// TIA Portal V19 export
FUNCTION_BLOCK "Coilcar_FB"   // FB96, LAD
TITLE = COIL CAR
// stored: MemoryReserve 100, SetENOAutomatically false
   VAR_INPUT
      AreaInterface : "AreaInterface";
      ZSI : "udt_ZoneSafetyInterface";
      DSI : Struct
         Move : "udt_DeviceSafetyInterface";
         LIft : "udt_DeviceSafetyInterface";
      END_STRUCT;
      Drive : "TAx_DriveInterface";
      HW_ID_TEL1 : HW_SUBMODULE;
      DataIn : Struct
         Supports_Ls_FixPoleLeft_Plugged : Bool;
         Supports_Ls_FixPoleRight_Plugged : Bool;
         Supports_Ls_MobilePoleLeft_Plugged : Bool;
         Supports_Ls_MobilePoleRight_Plugged : Bool;
         Move_Ls_Outline : Bool;
         Move_Ls_Inline : Bool;
         Move_Ls_LowSpeedOutline : Bool;
         Move_Ls_LowSpeedInline : Bool;
         Move_Ls_CoilInserted : Bool;   // TRUE = Movable supprts must be closed
         Move : "SpeedMachine_DataIn";
         Lift1 : "ValveMachine_DataIn";
         Lift2 : "ValveMachine_DataIn";
      END_STRUCT;
      CIn : Struct
         PressureRunning : Bool;
      END_STRUCT;
      Config : Struct
         LsStopDelayON { ExternalAccessible := 'False'; ExternalVisible := 'False'; ExternalWritable := 'False'} : Time := T#100ms;
         LsStopDelayOFF { ExternalAccessible := 'False'; ExternalVisible := 'False'; ExternalWritable := 'False'} : Time := T#200ms;
         Move : "SpeedMachine_Config";
         Lift1 : "ValveMachine_Config";
         Lift2 : "ValveMachine_Config";
      END_STRUCT;
   END_VAR
   VAR_OUTPUT
      MachineInterface : "MachineInterface";
      DataOut : Struct
         Move : "SpeedMachine_DataOut";
         Lift1 : "ValveMachine_DataOut";
         Lift2 : "ValveMachine_DataOut";
      END_STRUCT;
      COut : Struct
         IsInline : Bool;
         IsOutline : Bool;
         Move : "SpeedMachine_COut";
         Lift1 : "ValveMachine_COut";
         Lift2 : "ValveMachine_COut";
      END_STRUCT;
   END_VAR
   VAR_IN_OUT
      PersistentValues : Struct
         Move : "SpeedMachine_Par";
      END_STRUCT;
   END_VAR
   VAR
      Sts : Struct
         Move : Struct
            LowSpeedInline : Bool;
            LowSpeedOutline : Bool;
            IsInline : Bool;
            IsOutline : Bool;
            Inline_Cnd : Bool;
            Outline_Cnd : Bool;
            ReductionRatio : LReal;
         END_STRUCT;
         Free : Bool;
      END_STRUCT;
      Alarm : Struct
         Move_UnvalidStateLsInOut : Bool;
         Move_UnvalidStateLsLow : Bool;
         Move : "SpeedMachine_Alr";
         Lift1 : "ValveAlr";
         Lift2 : "ValveAlr";
      END_STRUCT;
      Warning : Struct
         Move : "SpeedMachine_Wng";
         Lift1 { ExternalAccessible := 'False'; ExternalVisible := 'False'; ExternalWritable := 'False'} : "ValveMachine_Wng";
         Lift2 { ExternalAccessible := 'False'; ExternalVisible := 'False'; ExternalWritable := 'False'} : "ValveMachine_Wng";
         NotOutline : Bool;
         Supports_FixPolesNotPlugged : Bool;
         Supports_MobilePolesNotPlugged : Bool;
      END_STRUCT;
      Move : "SpeedMachine_FB";
      Lift1 : "ValveMachine_FB";
      Lift2 : "ValveMachine_FB";
      TON_OutlinePos_DelayON : IEC_TIMER;
      TON_OutlinePos_DelayOFF : IEC_TIMER;
      TON_InlinePos_DelayON : IEC_TIMER;
      TON_InlinePos_DelayOFF : IEC_TIMER;
      pippo { S7_SetPoint := 'True'} : IEC_TIMER;
   END_VAR
   VAR_TEMP   // added for the SCL form of the ladder/FBD networks
      _w1 : Bool;
   END_VAR
BEGIN

REGION Network 1 (SCL): Reset alarms command

   IF  #AreaInterface.RstAlarms THEN
       // Alarms
       #Alarm.Move_UnvalidStateLsInOut := FALSE;
       #Alarm.Move_UnvalidStateLsLow := FALSE;



   END_IF;
END_REGION

REGION Network 2: >
END_REGION

REGION Network 3: <<< MOVE >>>
END_REGION

REGION Network 4: Alarm: Invalid state of inline/outline limit switches
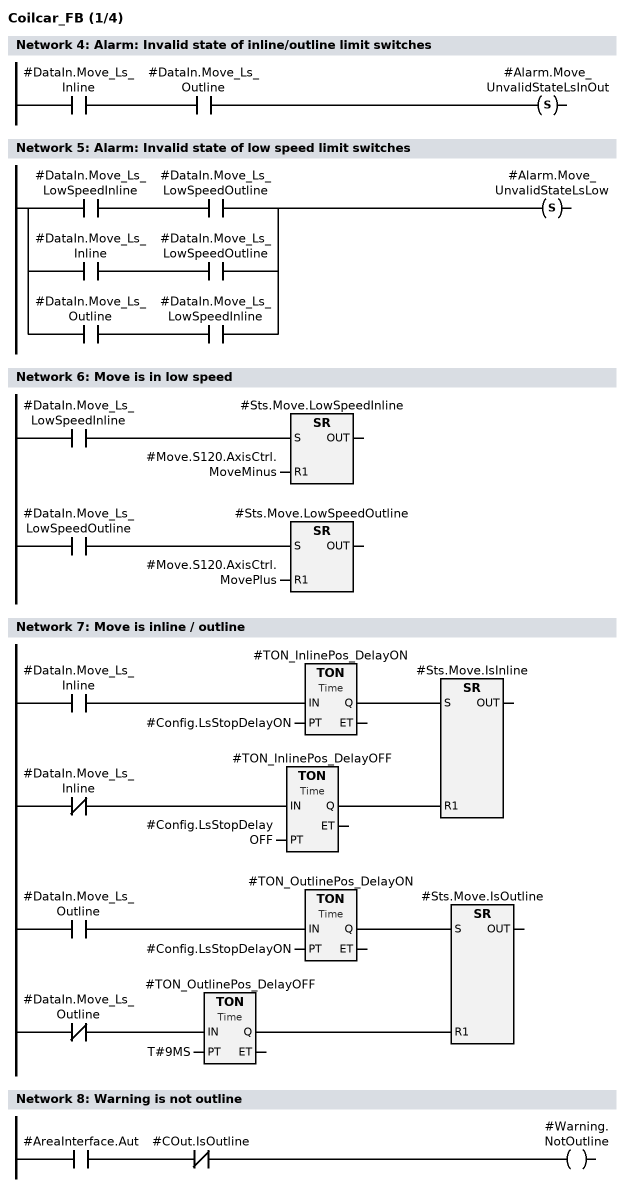
   RUNG wire#powerrail
      Contact( #DataIn.Move_Ls_Inline )
      Contact( #DataIn.Move_Ls_Outline )
      S_Coil( #Alarm.Move_UnvalidStateLsInOut )
   END_RUNG
   // the same network as SCL:
   IF #DataIn.Move_Ls_Inline AND #DataIn.Move_Ls_Outline THEN
       #Alarm.Move_UnvalidStateLsInOut := TRUE;
   END_IF;
END_REGION

REGION Network 5: Alarm: Invalid state of low speed limit switches
   RUNG wire#powerrail
      Contact( #DataIn.Move_Ls_LowSpeedInline )
      Contact( #DataIn.Move_Ls_LowSpeedOutline )
      wire#w1
      S_Coil( #Alarm.Move_UnvalidStateLsLow )
   END_RUNG
   RUNG wire#powerrail
      Contact( #DataIn.Move_Ls_Inline )
      Contact( #DataIn.Move_Ls_LowSpeedOutline )
   END_RUNG wire#w1
   RUNG wire#powerrail
      Contact( #DataIn.Move_Ls_Outline )
      Contact( #DataIn.Move_Ls_LowSpeedInline )
   END_RUNG wire#w1
   // the same network as SCL:
   IF (#DataIn.Move_Ls_LowSpeedInline AND #DataIn.Move_Ls_LowSpeedOutline) OR (#DataIn.Move_Ls_Inline AND #DataIn.Move_Ls_LowSpeedOutline) OR (#DataIn.Move_Ls_Outline AND #DataIn.Move_Ls_LowSpeedInline) THEN
       #Alarm.Move_UnvalidStateLsLow := TRUE;
   END_IF;
END_REGION

REGION Network 6: Move is in low speed
   RUNG wire#powerrail
      Contact( #DataIn.Move_Ls_LowSpeedInline )
      S_SR(operand := #Sts.Move.LowSpeedInline, r1 := #Move.S120.AxisCtrl.MoveMinus)
   END_RUNG
   RUNG wire#powerrail
      Contact( #DataIn.Move_Ls_LowSpeedOutline )
      S_SR(operand := #Sts.Move.LowSpeedOutline, r1 := #Move.S120.AxisCtrl.MovePlus)
   END_RUNG
   // the same network as SCL:
   IF #DataIn.Move_Ls_LowSpeedInline THEN
       #Sts.Move.LowSpeedInline := TRUE;   // SR flip-flop
   END_IF;
   IF #Move.S120.AxisCtrl.MoveMinus THEN #Sts.Move.LowSpeedInline := FALSE; END_IF;
   IF #DataIn.Move_Ls_LowSpeedOutline THEN
       #Sts.Move.LowSpeedOutline := TRUE;   // SR flip-flop
   END_IF;
   IF #Move.S120.AxisCtrl.MovePlus THEN #Sts.Move.LowSpeedOutline := FALSE; END_IF;
END_REGION

REGION Network 7: Move is inline / outline
   RUNG wire#powerrail
      Contact( #DataIn.Move_Ls_Inline )
      { S7_Templates := "time_type := Time" } #TON_InlinePos_DelayON.TON(pt := #Config.LsStopDelayON, et =>)
      S_SR(operand := #Sts.Move.IsInline, r1 := wire#w1)
   END_RUNG
   RUNG wire#powerrail
      I_Contact( #DataIn.Move_Ls_Inline )
      { S7_Templates := "time_type := Time" } #TON_InlinePos_DelayOFF.TON(pt := #Config.LsStopDelayOFF, et =>)
   END_RUNG wire#w1
   RUNG wire#powerrail
      Contact( #DataIn.Move_Ls_Outline )
      { S7_Templates := "time_type := Time" } #TON_OutlinePos_DelayON.TON(pt := #Config.LsStopDelayON, et =>)
      S_SR(operand := #Sts.Move.IsOutline, r1 := wire#w2)
   END_RUNG
   RUNG wire#powerrail
      I_Contact( #DataIn.Move_Ls_Outline )
      { S7_Templates := "time_type := Time" } #TON_OutlinePos_DelayOFF.TON(pt := T#9MS, et =>)
   END_RUNG wire#w2
   // the same network as SCL:
   #TON_InlinePos_DelayON.TON(IN := #DataIn.Move_Ls_Inline, PT := #Config.LsStopDelayON);
   #TON_InlinePos_DelayOFF.TON(IN := NOT #DataIn.Move_Ls_Inline, PT := #Config.LsStopDelayOFF);
   IF #TON_InlinePos_DelayON.Q THEN
       #Sts.Move.IsInline := TRUE;   // SR flip-flop
   END_IF;
   IF #TON_InlinePos_DelayOFF.Q THEN #Sts.Move.IsInline := FALSE; END_IF;
   #TON_OutlinePos_DelayON.TON(IN := #DataIn.Move_Ls_Outline, PT := #Config.LsStopDelayON);
   #TON_OutlinePos_DelayOFF.TON(IN := NOT #DataIn.Move_Ls_Outline, PT := T#9MS);
   IF #TON_OutlinePos_DelayON.Q THEN
       #Sts.Move.IsOutline := TRUE;   // SR flip-flop
   END_IF;
   IF #TON_OutlinePos_DelayOFF.Q THEN #Sts.Move.IsOutline := FALSE; END_IF;
END_REGION

REGION Network 8: Warning is not outline
   RUNG wire#powerrail
      Contact( #AreaInterface.Aut )
      I_Contact( #COut.IsOutline )
      Coil( #Warning.NotOutline )
   END_RUNG
   // the same network as SCL:
   #Warning.NotOutline := #AreaInterface.Aut AND NOT #COut.IsOutline;
END_REGION

REGION Network 9: Warnings for missing rotation conditions
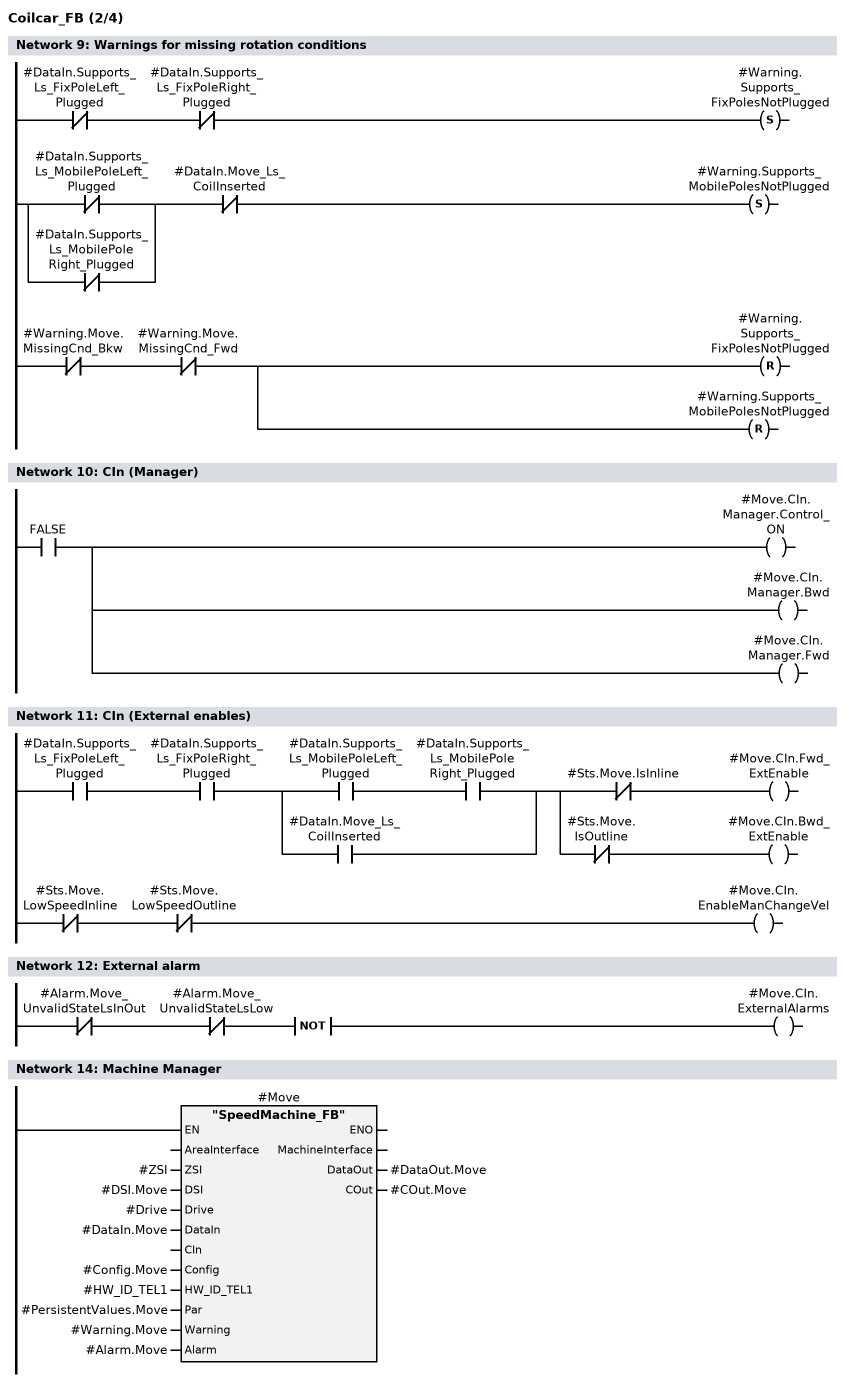
   RUNG wire#powerrail
      I_Contact( #DataIn.Supports_Ls_FixPoleLeft_Plugged )
      I_Contact( #DataIn.Supports_Ls_FixPoleRight_Plugged )
      S_Coil( #Warning.Supports_FixPolesNotPlugged )
   END_RUNG
   RUNG wire#powerrail
      I_Contact( #DataIn.Supports_Ls_MobilePoleLeft_Plugged )
      wire#w1
      I_Contact( #DataIn.Move_Ls_CoilInserted )
      S_Coil( #Warning.Supports_MobilePolesNotPlugged )
   END_RUNG
   RUNG wire#powerrail
      I_Contact( #DataIn.Supports_Ls_MobilePoleRight_Plugged )
   END_RUNG wire#w1
   RUNG wire#powerrail
      I_Contact( #Warning.Move.MissingCnd_Bkw )
      I_Contact( #Warning.Move.MissingCnd_Fwd )
      wire#w2
      R_Coil( #Warning.Supports_FixPolesNotPlugged )
   END_RUNG
   RUNG wire#w2
      R_Coil( #Warning.Supports_MobilePolesNotPlugged )
   END_RUNG
   // the same network as SCL:
   IF NOT #DataIn.Supports_Ls_FixPoleLeft_Plugged AND NOT #DataIn.Supports_Ls_FixPoleRight_Plugged THEN
       #Warning.Supports_FixPolesNotPlugged := TRUE;
   END_IF;
   IF (NOT #DataIn.Supports_Ls_MobilePoleLeft_Plugged OR NOT #DataIn.Supports_Ls_MobilePoleRight_Plugged) AND NOT #DataIn.Move_Ls_CoilInserted THEN
       #Warning.Supports_MobilePolesNotPlugged := TRUE;
   END_IF;
   IF NOT #Warning.Move.MissingCnd_Bkw AND NOT #Warning.Move.MissingCnd_Fwd THEN
       #Warning.Supports_FixPolesNotPlugged := FALSE;
       #Warning.Supports_MobilePolesNotPlugged := FALSE;
   END_IF;
END_REGION

REGION Network 10: CIn (Manager)
   RUNG wire#powerrail
      Contact( FALSE )
      wire#w1
      Coil( #Move.CIn.Manager.Control_ON )
   END_RUNG
   RUNG wire#w1
      Coil( #Move.CIn.Manager.Bwd )
   END_RUNG
   RUNG wire#w1
      Coil( #Move.CIn.Manager.Fwd )
   END_RUNG
   // the same network as SCL:
   #Move.CIn.Manager.Control_ON := FALSE;
   #Move.CIn.Manager.Bwd := FALSE;
   #Move.CIn.Manager.Fwd := FALSE;
END_REGION

REGION Network 11: CIn (External enables)
   RUNG wire#powerrail
      Contact( #DataIn.Supports_Ls_FixPoleLeft_Plugged )
      Contact( #DataIn.Supports_Ls_FixPoleRight_Plugged )
      wire#w1
      Contact( #DataIn.Supports_Ls_MobilePoleLeft_Plugged )
      Contact( #DataIn.Supports_Ls_MobilePoleRight_Plugged )
      wire#w2
      I_Contact( #Sts.Move.IsInline )
      Coil( #Move.CIn.Fwd_ExtEnable )
   END_RUNG
   RUNG wire#w1
      Contact( #DataIn.Move_Ls_CoilInserted )
   END_RUNG wire#w2
   RUNG wire#w2
      I_Contact( #Sts.Move.IsOutline )
      Coil( #Move.CIn.Bwd_ExtEnable )
   END_RUNG
   RUNG wire#powerrail
      I_Contact( #Sts.Move.LowSpeedInline )
      I_Contact( #Sts.Move.LowSpeedOutline )
      Coil( #Move.CIn.EnableManChangeVel )
   END_RUNG
   // the same network as SCL:
   #_w1 := #DataIn.Supports_Ls_FixPoleLeft_Plugged AND #DataIn.Supports_Ls_FixPoleRight_Plugged AND ((#DataIn.Supports_Ls_MobilePoleLeft_Plugged AND #DataIn.Supports_Ls_MobilePoleRight_Plugged) OR #DataIn.Move_Ls_CoilInserted);
   #Move.CIn.Fwd_ExtEnable := #_w1 AND NOT #Sts.Move.IsInline;
   #Move.CIn.Bwd_ExtEnable := #_w1 AND NOT #Sts.Move.IsOutline;
   #Move.CIn.EnableManChangeVel := NOT #Sts.Move.LowSpeedInline AND NOT #Sts.Move.LowSpeedOutline;
END_REGION

REGION Network 12: External alarm
   RUNG wire#powerrail
      I_Contact( #Alarm.Move_UnvalidStateLsInOut )
      I_Contact( #Alarm.Move_UnvalidStateLsLow )
      Not()
      Coil( #Move.CIn.ExternalAlarms )
   END_RUNG
   // the same network as SCL:
   #Move.CIn.ExternalAlarms := NOT (NOT #Alarm.Move_UnvalidStateLsInOut AND NOT #Alarm.Move_UnvalidStateLsLow);
END_REGION

REGION Network 13 (SCL): AreaInterface
   #Move.AreaInterface := #AreaInterface;

   #Move.AreaInterface.Man := #AreaInterface.Aut OR #AreaInterface.Man;
   #Move.AreaInterface.Aut := FALSE;
   #Move.AreaInterface.Cycle := FALSE;
END_REGION

REGION Network 14: Machine Manager
   RUNG wire#powerrail
      #Move(AreaInterface :=, ZSI := #ZSI, DSI := #DSI.Move, Drive := #Drive, DataIn := #DataIn.Move, CIn :=, Config := #Config.Move, HW_ID_TEL1 := #HW_ID_TEL1, Par := #PersistentValues.Move, Warning := #Warning.Move, Alarm := #Alarm.Move, MachineInterface =>, DataOut => #DataOut.Move, COut => #COut.Move)
   END_RUNG
   // the same network as SCL:
   #Move(ZSI := #ZSI,   // "SpeedMachine_FB"
         DSI := #DSI.Move,
         Drive := #Drive,
         DataIn := #DataIn.Move,
         Config := #Config.Move,
         HW_ID_TEL1 := #HW_ID_TEL1,
         Par := #PersistentValues.Move,
         Warning := #Warning.Move,
         Alarm := #Alarm.Move,
         DataOut => #DataOut.Move,
         COut => #COut.Move);
END_REGION

REGION Network 15: >
END_REGION

REGION Network 16: >
END_REGION

REGION Network 17: <<< LIFT 1 (REST = DOWN / WORK = UP)>>>
END_REGION

REGION Network 18: CIn (external enables)
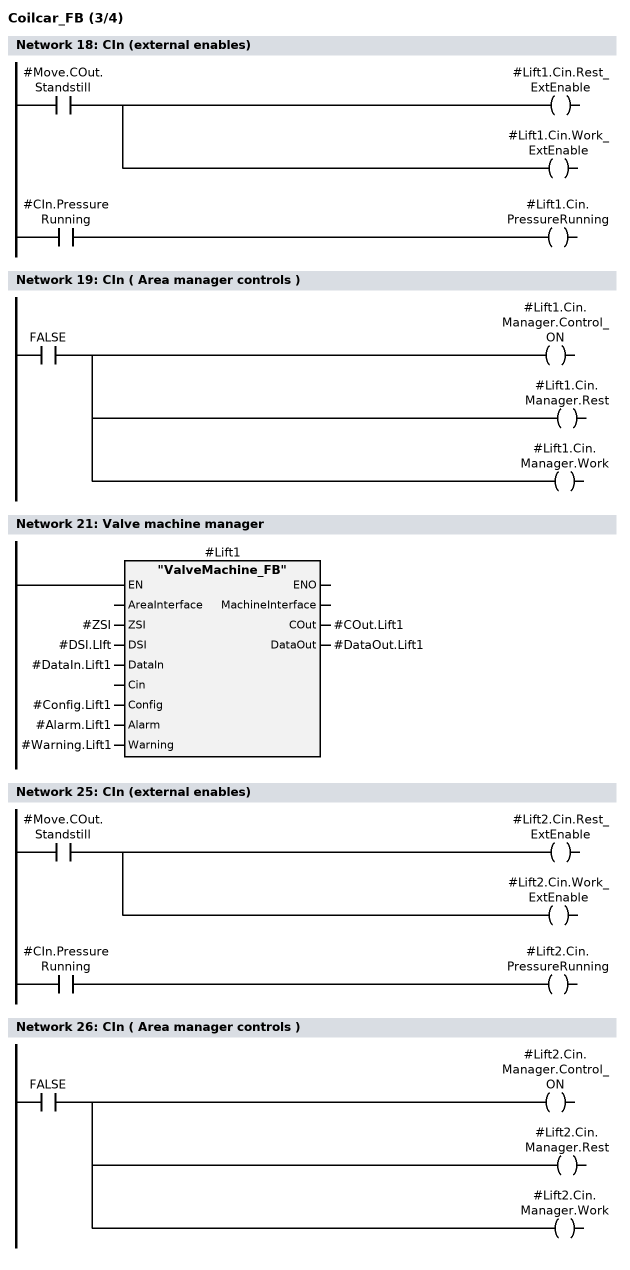
   RUNG wire#powerrail
      Contact( #Move.COut.Standstill )
      wire#w1
      Coil( #Lift1.Cin.Rest_ExtEnable )
   END_RUNG
   RUNG wire#w1
      Coil( #Lift1.Cin.Work_ExtEnable )
   END_RUNG
   RUNG wire#powerrail
      Contact( #CIn.PressureRunning )
      Coil( #Lift1.Cin.PressureRunning )
   END_RUNG
   // the same network as SCL:
   #Lift1.Cin.Rest_ExtEnable := #Move.COut.Standstill;
   #Lift1.Cin.Work_ExtEnable := #Move.COut.Standstill;
   #Lift1.Cin.PressureRunning := #CIn.PressureRunning;
END_REGION

REGION Network 19: CIn ( Area manager controls )
   RUNG wire#powerrail
      Contact( FALSE )
      wire#w1
      Coil( #Lift1.Cin.Manager.Control_ON )
   END_RUNG
   RUNG wire#w1
      Coil( #Lift1.Cin.Manager.Rest )
   END_RUNG
   RUNG wire#w1
      Coil( #Lift1.Cin.Manager.Work )
   END_RUNG
   // the same network as SCL:
   #Lift1.Cin.Manager.Control_ON := FALSE;
   #Lift1.Cin.Manager.Rest := FALSE;
   #Lift1.Cin.Manager.Work := FALSE;
END_REGION

REGION Network 20 (SCL): AreaInterface
   #Lift1.AreaInterface := #AreaInterface;

   #Lift1.AreaInterface.Man := #AreaInterface.Aut OR #AreaInterface.Man;
   #Lift1.AreaInterface.Aut := FALSE;
   #Lift1.AreaInterface.Cycle := FALSE;
END_REGION

REGION Network 21: Valve machine manager
   RUNG wire#powerrail
      #Lift1(AreaInterface :=, ZSI := #ZSI, DSI := #DSI.LIft, DataIn := #DataIn.Lift1, Cin :=, Config := #Config.Lift1, Alarm := #Alarm.Lift1, Warning := #Warning.Lift1, MachineInterface =>, COut => #COut.Lift1, DataOut => #DataOut.Lift1)
   END_RUNG
   // the same network as SCL:
   #Lift1(ZSI := #ZSI,   // "ValveMachine_FB"
          DSI := #DSI.LIft,
          DataIn := #DataIn.Lift1,
          Config := #Config.Lift1,
          Alarm := #Alarm.Lift1,
          Warning := #Warning.Lift1,
          COut => #COut.Lift1,
          DataOut => #DataOut.Lift1);
END_REGION

REGION Network 22: >
END_REGION

REGION Network 23: >
END_REGION

REGION Network 24: <<< LIFT 1 (REST = DOWN / WORK = UP)>>>
END_REGION

REGION Network 25: CIn (external enables)
   RUNG wire#powerrail
      Contact( #Move.COut.Standstill )
      wire#w1
      Coil( #Lift2.Cin.Rest_ExtEnable )
   END_RUNG
   RUNG wire#w1
      Coil( #Lift2.Cin.Work_ExtEnable )
   END_RUNG
   RUNG wire#powerrail
      Contact( #CIn.PressureRunning )
      Coil( #Lift2.Cin.PressureRunning )
   END_RUNG
   // the same network as SCL:
   #Lift2.Cin.Rest_ExtEnable := #Move.COut.Standstill;
   #Lift2.Cin.Work_ExtEnable := #Move.COut.Standstill;
   #Lift2.Cin.PressureRunning := #CIn.PressureRunning;
END_REGION

REGION Network 26: CIn ( Area manager controls )
   RUNG wire#powerrail
      Contact( FALSE )
      wire#w1
      Coil( #Lift2.Cin.Manager.Control_ON )
   END_RUNG
   RUNG wire#w1
      Coil( #Lift2.Cin.Manager.Rest )
   END_RUNG
   RUNG wire#w1
      Coil( #Lift2.Cin.Manager.Work )
   END_RUNG
   // the same network as SCL:
   #Lift2.Cin.Manager.Control_ON := FALSE;
   #Lift2.Cin.Manager.Rest := FALSE;
   #Lift2.Cin.Manager.Work := FALSE;
END_REGION

REGION Network 27 (SCL): AreaInterface
   #Lift2.AreaInterface := #AreaInterface;

   #Lift2.AreaInterface.Man := #AreaInterface.Aut OR #AreaInterface.Man;
   #Lift2.AreaInterface.Aut := FALSE;
   #Lift2.AreaInterface.Cycle := FALSE;
END_REGION

REGION Network 28: Valve machine manager
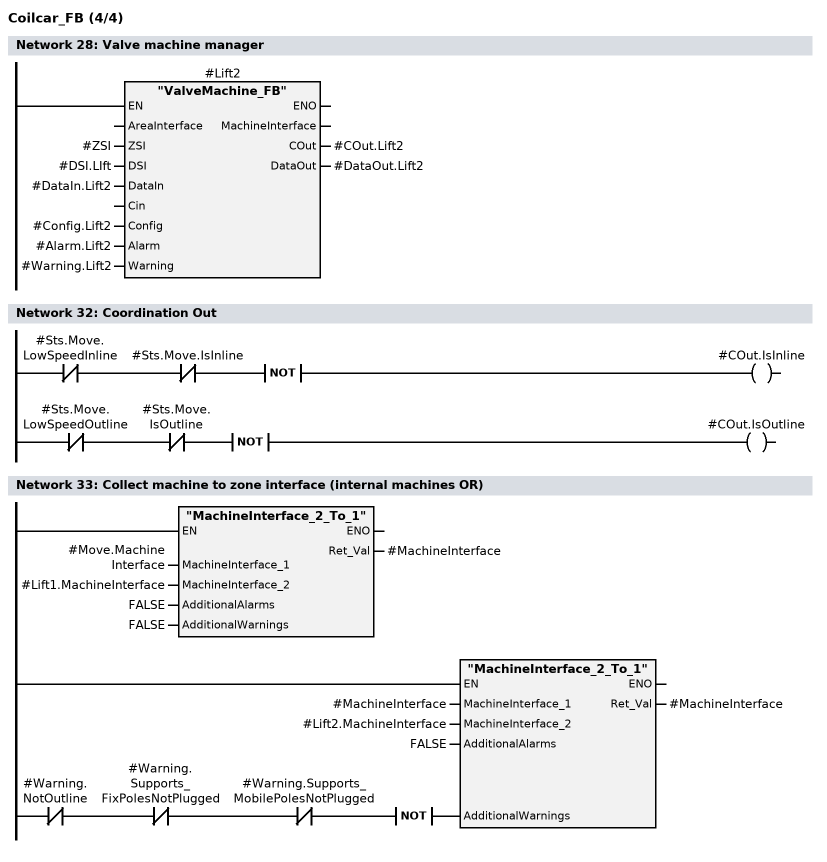
   RUNG wire#powerrail
      #Lift2(AreaInterface :=, ZSI := #ZSI, DSI := #DSI.LIft, DataIn := #DataIn.Lift2, Cin :=, Config := #Config.Lift2, Alarm := #Alarm.Lift2, Warning := #Warning.Lift2, MachineInterface =>, COut => #COut.Lift2, DataOut => #DataOut.Lift2)
   END_RUNG
   // the same network as SCL:
   #Lift2(ZSI := #ZSI,   // "ValveMachine_FB"
          DSI := #DSI.LIft,
          DataIn := #DataIn.Lift2,
          Config := #Config.Lift2,
          Alarm := #Alarm.Lift2,
          Warning := #Warning.Lift2,
          COut => #COut.Lift2,
          DataOut => #DataOut.Lift2);
END_REGION

REGION Network 29: >
END_REGION

REGION Network 30: >
END_REGION

REGION Network 31: <<< MACHINE STATUS >>>
END_REGION

REGION Network 32: Coordination Out
   RUNG wire#powerrail
      I_Contact( #Sts.Move.LowSpeedInline )
      I_Contact( #Sts.Move.IsInline )
      Not()
      Coil( #COut.IsInline )
   END_RUNG
   RUNG wire#powerrail
      I_Contact( #Sts.Move.LowSpeedOutline )
      I_Contact( #Sts.Move.IsOutline )
      Not()
      Coil( #COut.IsOutline )
   END_RUNG
   // the same network as SCL:
   #COut.IsInline := NOT (NOT #Sts.Move.LowSpeedInline AND NOT #Sts.Move.IsInline);
   #COut.IsOutline := NOT (NOT #Sts.Move.LowSpeedOutline AND NOT #Sts.Move.IsOutline);
END_REGION

REGION Network 33: Collect machine to zone interface (internal machines OR)
   RUNG wire#powerrail
      "MachineInterface_2_To_1"(MachineInterface_1 := #Move.MachineInterface, MachineInterface_2 := #Lift1.MachineInterface, AdditionalAlarms := FALSE, AdditionalWarnings := FALSE, Ret_Val => #MachineInterface)
   END_RUNG
   RUNG wire#powerrail
      "MachineInterface_2_To_1"(AdditionalWarnings := wire#w1, MachineInterface_1 := #MachineInterface, MachineInterface_2 := #Lift2.MachineInterface, AdditionalAlarms := FALSE, Ret_Val => #MachineInterface)
   END_RUNG
   RUNG wire#powerrail
      I_Contact( #Warning.NotOutline )
      I_Contact( #Warning.Supports_FixPolesNotPlugged )
      I_Contact( #Warning.Supports_MobilePolesNotPlugged )
      Not()
   END_RUNG wire#w1
   // the same network as SCL:
   #MachineInterface := "MachineInterface_2_To_1"(MachineInterface_1 := #Move.MachineInterface,
                           MachineInterface_2 := #Lift1.MachineInterface,
                           AdditionalAlarms := FALSE,
                           AdditionalWarnings := FALSE);
   #MachineInterface := "MachineInterface_2_To_1"(MachineInterface_1 := #MachineInterface,
                           MachineInterface_2 := #Lift2.MachineInterface,
                           AdditionalAlarms := FALSE,
                           AdditionalWarnings := NOT (NOT #Warning.NotOutline AND NOT #Warning.Supports_FixPolesNotPlugged AND NOT #Warning.Supports_MobilePolesNotPlugged));
END_REGION

REGION Network 34: >
END_REGION

REGION Network 35: >
END_REGION
END_FUNCTION_BLOCK
